PROGRAM RunGrindingWell
VAR
END_VAR

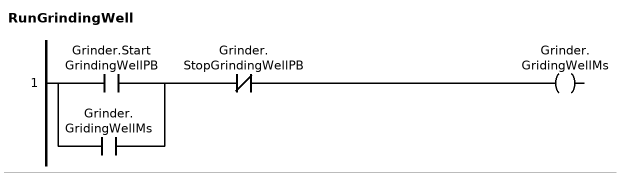
// NETWORK 1
Grinder.GridingWellMs := (Grinder.StartGrindingWellPB OR Grinder.GridingWellMs) AND NOT Grinder.StopGrindingWellPB;

END_PROGRAM

(* stored: Version 1.1.0.1, ProductVersion 3.1.4024.4
   POU RunGrindingWell: Id {cc4cedd0-9202-4fc8-aaf2-e05dc1c13db3}, SpecialFunc None *)
